SYSTEM ReferenceExamples
  (* Version 1.0, 2022-06-27, AK115394 *)
  APPLICATION _01_EventConnections
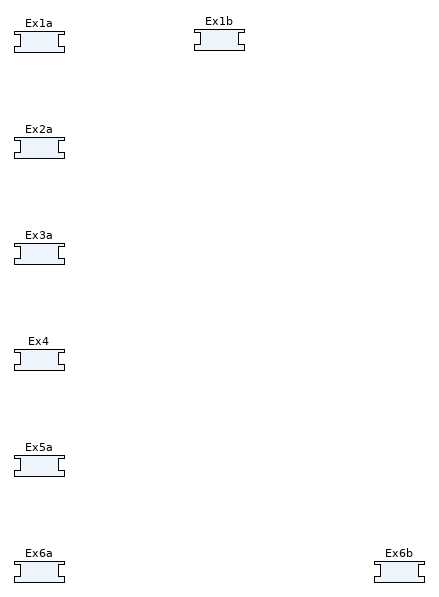
    (* Group Info_EventConnections: The subapps in this App serve as test cases for various versions of event connections: &#10;- simple connections &#10;- fan-out &#10;- fan-in  &#10;- self-loop &#10;- connections between different kinds of FBs &#10;- a loop (repeated event connection use) &#10; *)
    SUBAPPLICATION Ex1a (* simple event connection  &#10;- trigger E_SPLIT.EI  &#10;- expect E_REND.EO *)
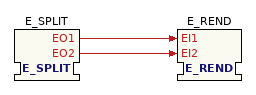
      FBS
        E_SPLIT : E_SPLIT;
        E_REND : E_REND;
      END_FBS
      EVENT_CONNECTIONS
        E_SPLIT.EO1 TO E_REND.EI1;
        E_SPLIT.EO2 TO E_REND.EI2;
      END_CONNECTIONS
    END_SUBAPPLICATION
    SUBAPPLICATION Ex1b (* simple event connection across several FBs   &#10;- trigger E_SPLIT.EI    &#10;- expect E_REND.EO and &#10;   E_SPLIT2.EO1 and E_SPLIT2.EO2 *)
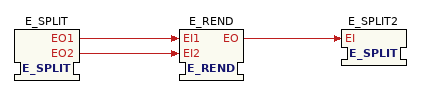
      FBS
        E_SPLIT : E_SPLIT;
        E_SPLIT2 : E_SPLIT;
        E_REND : E_REND;
      END_FBS
      EVENT_CONNECTIONS
        E_SPLIT.EO1 TO E_REND.EI1;
        E_SPLIT.EO2 TO E_REND.EI2;
        E_REND.EO TO E_SPLIT2.EI;
      END_CONNECTIONS
    END_SUBAPPLICATION
    SUBAPPLICATION Ex5a (* example involving simple FB and basic FB type &#10;- trigger E_PERMIT.EI &#10;- expect SimpleIO.CNF, DOI1 := TRUE *)
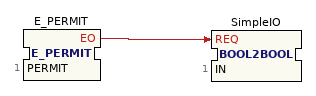
      FBS
        E_PERMIT : E_PERMIT(PERMIT := 1);
        SimpleIO : BOOL2BOOL(IN := 1);
      END_FBS
      EVENT_CONNECTIONS
        E_PERMIT.EO TO SimpleIO.REQ;
      END_CONNECTIONS
    END_SUBAPPLICATION
    SUBAPPLICATION Ex2a (* fan-out of event connections  &#10;- trigger E_SPLIT.EI  &#10;- expect 2xE_MERGE.EO *)
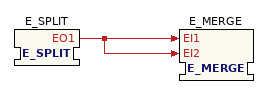
      FBS
        E_SPLIT : E_SPLIT;
        E_MERGE : E_MERGE;
      END_FBS
      EVENT_CONNECTIONS
        E_SPLIT.EO1 TO E_MERGE.EI1;
        E_SPLIT.EO1 TO E_MERGE.EI2;
      END_CONNECTIONS
    END_SUBAPPLICATION
    SUBAPPLICATION Ex3a (* fan-in of event connections  &#10;- trigger E_SPLIT.EI  &#10;- expect 2x E_CTU.CUO, CV := 2, Q:= TRUE *)
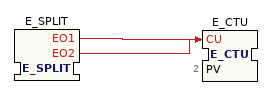
      FBS
        E_SPLIT : E_SPLIT;
        E_CTU : E_CTU(PV := 2);
      END_FBS
      EVENT_CONNECTIONS
        E_SPLIT.EO1 TO E_CTU.CU;
        E_SPLIT.EO2 TO E_CTU.CU;
      END_CONNECTIONS
    END_SUBAPPLICATION
    SUBAPPLICATION Ex6a (* for loop  &#10;- trigger 1x E_PERMIT.EI  &#10;- expect 2x CUO and 2x SimpleNOT.CNF and CV := 2 *)
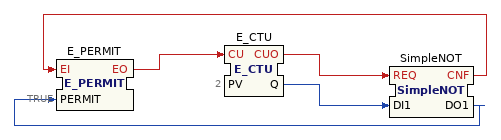
      FBS
        E_PERMIT : E_PERMIT(PERMIT := TRUE);
        E_CTU : E_CTU(PV := 2);
        SimpleNOT : SimpleNOT;
      END_FBS
      EVENT_CONNECTIONS
        E_PERMIT.EO TO E_CTU.CU;
        E_CTU.CUO TO SimpleNOT.REQ;
        SimpleNOT.CNF TO E_PERMIT.EI;
      END_CONNECTIONS
      DATA_CONNECTIONS
        E_CTU.Q TO SimpleNOT.DI1;
        SimpleNOT.DO1 TO E_PERMIT.PERMIT;
      END_CONNECTIONS
    END_SUBAPPLICATION
    SUBAPPLICATION Ex6b (* for loop  &#10;- trigger 1x E_PERMIT.EI  &#10;- expect no outputs *)
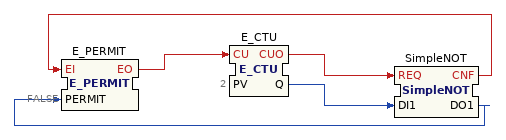
      FBS
        E_PERMIT : E_PERMIT(PERMIT := FALSE);
        E_CTU : E_CTU(PV := 2);
        SimpleNOT : SimpleNOT;
      END_FBS
      EVENT_CONNECTIONS
        E_PERMIT.EO TO E_CTU.CU;
        E_CTU.CUO TO SimpleNOT.REQ;
        SimpleNOT.CNF TO E_PERMIT.EI;
      END_CONNECTIONS
      DATA_CONNECTIONS
        E_CTU.Q TO SimpleNOT.DI1;
        SimpleNOT.DO1 TO E_PERMIT.PERMIT;
      END_CONNECTIONS
    END_SUBAPPLICATION
    SUBAPPLICATION Ex4 (* self-loop  &#10;- trigger E_CTU.R   &#10;- expect RO -&gt; CUO (CV:=1) *)
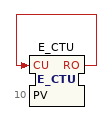
      FBS
        E_CTU : E_CTU(PV := 10);
      END_FBS
      EVENT_CONNECTIONS
        E_CTU.RO TO E_CTU.CU;
      END_CONNECTIONS
    END_SUBAPPLICATION
  END_APPLICATION
  APPLICATION _03_DataConnections
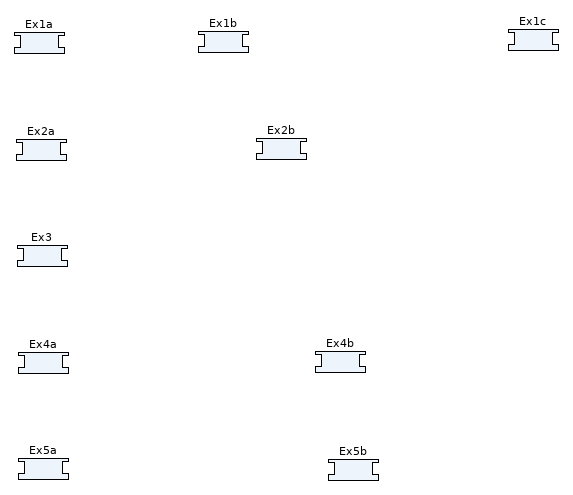
    (* Group Info_DataConnections: The subapps in this App serve as test cases for various versions of parameters: &#10;- simple boolean parameters (including counter-examples) &#10;- initial value taken from type when no parameter is present &#10;- parameters with prefixes &#10;- upcasts in parameters *)
    SUBAPPLICATION Ex2a (* fan-out of data connections &#10;- trigger Fb1.REQ &#10;- expect Fb2a.CNF with FB2a.OUT := TRUE AND Fb2b.CNF with FB2b.OUT *)
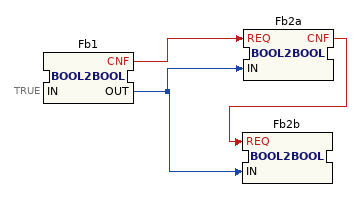
      FBS
        Fb1 : BOOL2BOOL(IN := TRUE);
        Fb2a : BOOL2BOOL;
        Fb2b : BOOL2BOOL;
      END_FBS
      EVENT_CONNECTIONS
        Fb1.CNF TO Fb2a.REQ;
        Fb2a.CNF TO Fb2b.REQ;
      END_CONNECTIONS
      DATA_CONNECTIONS
        Fb1.OUT TO Fb2a.IN;
        Fb1.OUT TO Fb2b.IN;
      END_CONNECTIONS
    END_SUBAPPLICATION
    SUBAPPLICATION Ex3 (* example involving two kinds of FB types (simple FB type and basic FB type)  &#10;trigger E_SR.S  &#10;expect SimpleIO.CNF, DOI1 := TRUE *)
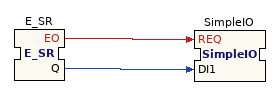
      FBS
        E_SR : E_SR;
        SimpleIO : SimpleIO;
      END_FBS
      EVENT_CONNECTIONS
        E_SR.EO TO SimpleIO.REQ;
      END_CONNECTIONS
      DATA_CONNECTIONS
        E_SR.Q TO SimpleIO.DI1;
      END_CONNECTIONS
    END_SUBAPPLICATION
    SUBAPPLICATION Ex4a (* type casts (explicit, upcast)  &#10;- trigger Fb1.CU  &#10;- expect Fb3.CNF and Fb3.OUT:=INT#1 *)
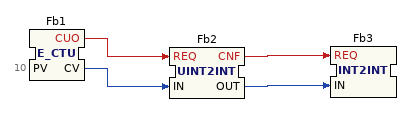
      FBS
        Fb1 : E_CTU(PV := 10);
        Fb3 : INT2INT;
        Fb2 : UINT2INT;
      END_FBS
      EVENT_CONNECTIONS
        Fb1.CUO TO Fb2.REQ;
        Fb2.CNF TO Fb3.REQ;
      END_CONNECTIONS
      DATA_CONNECTIONS
        Fb1.CV TO Fb2.IN;
        Fb2.OUT TO Fb3.IN;
      END_CONNECTIONS
    END_SUBAPPLICATION
    SUBAPPLICATION Ex1a (* simple data connection (BOOL) &#10;- trigger Fb1.REQ &#10;- expect Fb2.CNF with Fb2.OUT:=TRUE *)
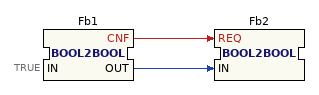
      FBS
        Fb1 : BOOL2BOOL(IN := TRUE);
        Fb2 : BOOL2BOOL;
      END_FBS
      EVENT_CONNECTIONS
        Fb1.CNF TO Fb2.REQ;
      END_CONNECTIONS
      DATA_CONNECTIONS
        Fb1.OUT TO Fb2.IN;
      END_CONNECTIONS
    END_SUBAPPLICATION
    SUBAPPLICATION Ex1b (* simple data connection (INT) &#10;- trigger Fb1.REQ &#10;- expect Fb2.CNF with Fb2.OUT:=5 *)
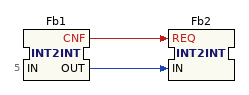
      FBS
        Fb1 : INT2INT(IN := 5);
        Fb2 : INT2INT;
      END_FBS
      EVENT_CONNECTIONS
        Fb1.CNF TO Fb2.REQ;
      END_CONNECTIONS
      DATA_CONNECTIONS
        Fb1.OUT TO Fb2.IN;
      END_CONNECTIONS
    END_SUBAPPLICATION
    SUBAPPLICATION Ex1c (* simple data connection (WORD) &#10;- trigger Fb1.REQ &#10;- expect Fb2.CNF with Fb2.OUT:=AFFE *)
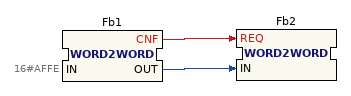
      FBS
        Fb1 : WORD2WORD(IN := 16#AFFE);
        Fb2 : WORD2WORD;
      END_FBS
      EVENT_CONNECTIONS
        Fb1.CNF TO Fb2.REQ;
      END_CONNECTIONS
      DATA_CONNECTIONS
        Fb1.OUT TO Fb2.IN;
      END_CONNECTIONS
    END_SUBAPPLICATION
    SUBAPPLICATION Ex2b (* fan-out of data connections &#10;- trigger Fb1.REQ &#10;- expect Fb2a.CNF with FB2a.OUT := TRUE AND Fb2b.CNF with FB2b.OUT:=TRUE AND  &#10;Fb2c.CNF with FB2c.OUT:=TRUE *)
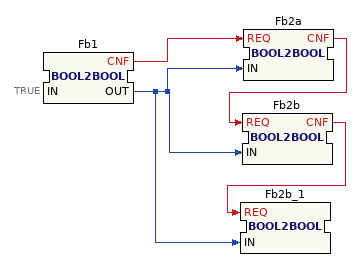
      FBS
        Fb1 : BOOL2BOOL(IN := TRUE);
        Fb2a : BOOL2BOOL;
        Fb2b : BOOL2BOOL;
        Fb2b_1 : BOOL2BOOL;
      END_FBS
      EVENT_CONNECTIONS
        Fb1.CNF TO Fb2a.REQ;
        Fb2a.CNF TO Fb2b.REQ;
        Fb2b.CNF TO Fb2b_1.REQ;
      END_CONNECTIONS
      DATA_CONNECTIONS
        Fb1.OUT TO Fb2a.IN;
        Fb1.OUT TO Fb2b.IN;
        Fb1.OUT TO Fb2b_1.IN;
      END_CONNECTIONS
    END_SUBAPPLICATION
    SUBAPPLICATION Ex4b (* type casts (explicit, downcast) &#10;- trigger Fb1.REQ &#10;- expect Fb3.CUO and CV:=1 and Q:=TRUE *)
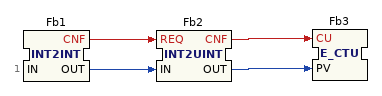
      FBS
        Fb1 : INT2INT(IN := 1);
        Fb3 : E_CTU;
        Fb2 : INT2UINT;
      END_FBS
      EVENT_CONNECTIONS
        Fb1.CNF TO Fb2.REQ;
        Fb2.CNF TO Fb3.CU;
      END_CONNECTIONS
      DATA_CONNECTIONS
        Fb1.OUT TO Fb2.IN;
        Fb2.OUT TO Fb3.PV;
      END_CONNECTIONS
    END_SUBAPPLICATION
    SUBAPPLICATION Ex5a (* type casts (implicit, upcast from UINT to ANY_MAG) &#10;- trigger Fb1.CU &#10;- expect Fb2.CNF and Fb2.OUT:=INT#6 *)
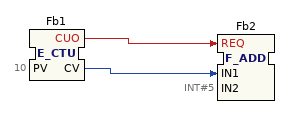
      FBS
        Fb1 : E_CTU(PV := 10);
        Fb2 : F_ADD(IN2 := INT#5);
      END_FBS
      EVENT_CONNECTIONS
        Fb1.CUO TO Fb2.REQ;
      END_CONNECTIONS
      DATA_CONNECTIONS
        Fb1.CV TO Fb2.IN1;
      END_CONNECTIONS
    END_SUBAPPLICATION
    SUBAPPLICATION Ex5b (* type casts (implicit, upcast from UINT to ANY_MAG) &#10;- trigger Fb1.CU &#10;- expect Fb2.CNF and Fb2.OUT:=REAL#1.0 *)
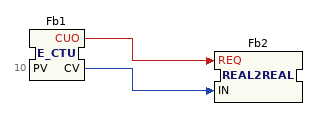
      FBS
        Fb1 : E_CTU(PV := 10);
        Fb2 : REAL2REAL;
      END_FBS
      EVENT_CONNECTIONS
        Fb1.CUO TO Fb2.REQ;
      END_CONNECTIONS
      DATA_CONNECTIONS
        Fb1.CV TO Fb2.IN;
      END_CONNECTIONS
    END_SUBAPPLICATION
  END_APPLICATION
  APPLICATION _07_Subapplications
    (* Group __Group01: connection to the interface *)
  END_APPLICATION
  APPLICATION _06_CompositeFBs
    (* Group __Group01: WITH bei composite FBs *)
  END_APPLICATION
  APPLICATION _02_Parameters
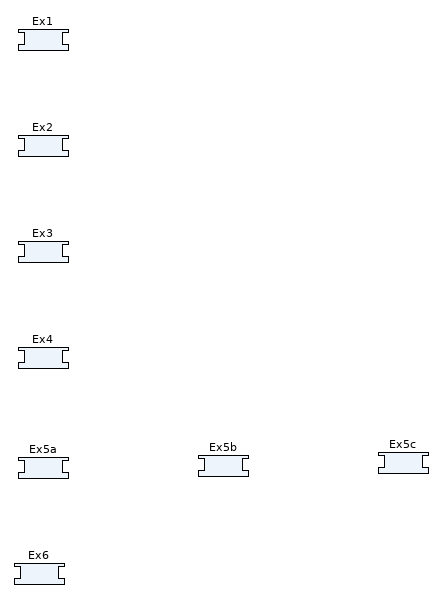
    (* Group Info_Parameters: The subapps in this App serve as test cases for various versions of parameters: &#10;- simple boolean parameters (including counter-examples) &#10;- initial value taken from type when no parameter is present &#10;- parameters with prefixes &#10;- upcasts in parameters *)
    SUBAPPLICATION Ex2 (* Parameters &#10; &#10;- Trigger EI  &#10;- Expect nothing *)
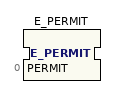
      FBS
        E_PERMIT : E_PERMIT(PERMIT := 0);
      END_FBS
    END_SUBAPPLICATION
    SUBAPPLICATION Ex1 (* Parameters overriding initial value of data type &#10; &#10;- Trigger E_PERMIT.EI  &#10;- Expect E_PERMIT.EO *)
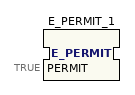
      FBS
        E_PERMIT_1 : E_PERMIT(PERMIT := TRUE);
      END_FBS
    END_SUBAPPLICATION
    SUBAPPLICATION Ex3 (* Initial Value (from type) &#10; &#10;- Trigger EI  &#10;- Expect EO *)
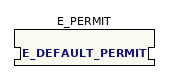
      FBS
        E_PERMIT : E_DEFAULT_PERMIT;
      END_FBS
    END_SUBAPPLICATION
    SUBAPPLICATION Ex4 (* Override initial value (from type) with parameter &#10; &#10;- Trigger EI  &#10;- Expect nothing *)
